INTERFACE I_Track

METHOD Clear : BOOL
VAR_INPUT
END_VAR
END_METHOD

METHOD Cycle : BOOL
VAR_INPUT
END_VAR
END_METHOD

METHOD Initialize : BOOL
VAR_INPUT
	nTrackIndex	: UDINT;
END_VAR
END_METHOD

PROPERTY P_Error : Bool
GET
END_GET
END_PROPERTY

PROPERTY P_TrackLength : LREAL
GET
END_GET
END_PROPERTY

PROPERTY std : I_TrackStandard
GET
END_GET
END_PROPERTY

END_INTERFACE

(* stored: Version 1.1.0.1
   Itf I_Track: Id {20038d1a-3084-4988-90ae-edbc9e998b79}
   Method Clear: Id {b35f5f98-fb5f-4712-970e-18873dfdb214}
   Method Cycle: Id {2a9a3ab4-9667-4b08-b35b-9ca5e49a5470}
   Method Initialize: Id {78ad5bf6-329e-4f08-9471-200afd1c518b}
   Property P_Error: Id {d9ae669a-1d92-4c73-be6a-22b7bc9bde8b}
   Get Get: Id {93bc8f88-214b-4500-8443-cb53712e5395}
   Property P_TrackLength: Id {665ede21-68c2-4d48-93a4-89b98c5172b5}
   Get Get: Id {1e51982a-ba69-4db8-bb2b-25abb189bdfe}
   Property std: Id {147ccd20-c2c5-4dad-a5ba-c20c057326a2}
   Get Get: Id {ec0e9cb1-4f66-41b2-b659-9e5b14ad902c} *)
